// TIA Portal V16 program export: 1 tag tables, 1 data types, 3 data blocks, 9 code blocks (in call order from the OBs), 2 instance data blocks

VAR_GLOBAL   // PLC tag table "Default tag table"
   System_Byte AT %MB1 : Byte;
   FirstScan AT %M1.0 : Bool;
   DiagStatusUpdate AT %M1.1 : Bool;
   AlwaysTRUE AT %M1.2 : Bool;
   AlwaysFALSE AT %M1.3 : Bool;
   Clock_Byte AT %MB0 : Byte;
   Clock_10Hz AT %M0.0 : Bool;
   Clock_5Hz AT %M0.1 : Bool;
   "Clock_2.5Hz" AT %M0.2 : Bool;
   Clock_2Hz AT %M0.3 : Bool;
   "Clock_1.25Hz" AT %M0.4 : Bool;
   Clock_1Hz AT %M0.5 : Bool;
   "Clock_0.625Hz" AT %M0.6 : Bool;
   "Clock_0.5Hz" AT %M0.7 : Bool;
   PositioningAxis_1_Actor_Interface_AddressIn AT %I0.0 : "PD_TEL105_IN";
   PositioningAxis_1_Actor_Interface_AddressOut AT %Q0.0 : "PD_TEL105_OUT";
   PositioningAxis_1_Actor_Interface_TorqueDataAddressIn AT %I40.0 : "PD_TEL750_IN";
   PositioningAxis_1_Actor_Interface_TorqueDataAddressOut AT %Q40.0 : "PD_TEL750_OUT";
   "PositioningAxis_1_Actor_Interface_TorqueDataAddressIn(1)" AT %I44.0 : "PD_TEL750_IN";
   "PositioningAxis_1_Actor_Interface_TorqueDataAddressOut(1)" AT %Q52.0 : "PD_TEL750_OUT";
   SynchronousAxis_1_Actor_Interface_AddressIn AT %I20.0 : "PD_TEL105_IN";
   SynchronousAxis_1_Actor_Interface_AddressOut AT %Q20.0 : "PD_TEL105_OUT";
   SynchronousAxis_1_Actor_Interface_TorqueDataAddressIn AT %I42.0 : "PD_TEL750_IN";
   SynchronousAxis_1_Actor_Interface_TorqueDataAddressOut AT %Q46.0 : "PD_TEL750_OUT";
   "SynchronousAxis_1_Actor_Interface_TorqueDataAddressIn(1)" AT %I46.0 : "PD_TEL750_IN";
   "SynchronousAxis_1_Actor_Interface_TorqueDataAddressOut(1)" AT %Q58.0 : "PD_TEL750_OUT";
END_VAR

TYPE "quad_cnst_array"
// stored: IsFailsafeCompliant false
   STRUCT
      element : Array[0..3, 0..2] of Real;
   END_STRUCT;
   // element[0,0] := 0.00415;   // a
   // element[0,1] := 0.452;   // b
   // element[0,2] := 330.0;   // c
   // element[1,0] := -8.44E-07;   // a
   // element[1,1] := 0.000463;   // b
   // element[1,2] := 0.791;   // c
   // element[2,0] := -9.35E-05;   // a
   // element[2,1] := 0.000775;   // b
   // element[2,2] := 6.34;   // c
   // element[3,0] := -9.04E-05;   // a
   // element[3,1] := 0.0284;   // b
   // element[3,2] := 1.09;   // c
END_TYPE

DATA_BLOCK "testing_purposes"   // DB2
{ S7_Optimized_Access := 'TRUE' }
VERSION : 0.1
// stored: AutoNumber true, DBAccessibleFromOPCUA true, IsOnlyStoredInLoadMemory false, IsRetainMemResEnabled false, IsWriteProtectedInAS false, MemoryReserve 100
   VAR
      emc_calculated : Real;   // EMC_returned
      Temperature : Real := 20.0;   // Chamber temperature [C]
      Air_humi : Real;   // Air humidity [%]
      TemperatureWet : Real := 15.0;   // Wet bulb temperature [C]
      Air_humi_calc : Real;   // Calculated air humidity [%]
      TemperatureWet_calc : Real;   // Calculated wet bulb temperature [C]
      real_sig : Real := 0.0;
      real_win_len : UInt := 20;
      filt_real_sig : Real;
      real_ret_result : Int;   // Real filter work result
      lreal_sig : Real := 0.0;
      lreal_win_len : UInt := 30;
      filt_lreal_sig : Real;
      lreal_ret_result : Int;   // lReal filter work result
   END_VAR
BEGIN
END_DATA_BLOCK

DATA_BLOCK "air_data"   // DB1
{ S7_Optimized_Access := 'TRUE' }
VERSION : 0.1
// stored: AutoNumber true, DBAccessibleFromOPCUA true, IsOnlyStoredInLoadMemory false, IsRetainMemResEnabled false, IsWriteProtectedInAS false, MemoryReserve 100
   VAR RETAIN
      calc_const { S7_SetPoint := 'True'} : "quad_cnst_array";
      Pmean { S7_SetPoint := 'True'} : Real := 1013.25;   // Mean atmospheric pressure [hPa] (mbar)
   END_VAR
BEGIN
END_DATA_BLOCK

DATA_BLOCK "test_blocks_parameters"   // DB4
{ S7_Optimized_Access := 'TRUE' }
VERSION : 0.1
// stored: AutoNumber true, DBAccessibleFromOPCUA true, IsOnlyStoredInLoadMemory false, IsRetainMemResEnabled false, IsWriteProtectedInAS false, MemoryReserve 100
   VAR
      enable : Bool;
      Reset : Bool;
      Restart_to : Bool;
      Home : Bool;
      Settings : Struct
         HomeMode : Int;
      END_STRUCT;
   END_VAR
BEGIN
END_DATA_BLOCK

ORGANIZATION_BLOCK "Main"   // OB1, LAD, ProgramCycle
TITLE = "Main Program Sweep (Cycle)"
{ S7_Optimized_Access := 'TRUE' }
VERSION : 0.1
// stored: AutoNumber true, IsIECCheckEnabled false, SetENOAutomatically false
   VAR_INPUT
      Initial_Call : Bool;   // Initial call of this OB
      Remanence : Bool;   // =True, if remanent data are available
   END_VAR
BEGIN

REGION Network 2 (SCL)
   "test_blocks_DB"();
END_REGION
END_ORGANIZATION_BLOCK

FUNCTION_BLOCK "test_blocks"   // FB2, LAD
{ S7_Optimized_Access := 'TRUE' }
VERSION : 0.1
// stored: AutoNumber true, IsIECCheckEnabled false, IsRetainMemResEnabled false, MemoryReserve 100, SetENOAutomatically false, UDAEnableTagReadback false
   VAR
      MC_POWER_Instance { S7_SetPoint := 'True'} : MC_POWER;
      MC_RESET_Instance { S7_SetPoint := 'True'} : MC_RESET;
      MC_HOME_Instance { S7_SetPoint := 'True'} : MC_HOME;
   END_VAR
BEGIN

REGION Network 1: Enable
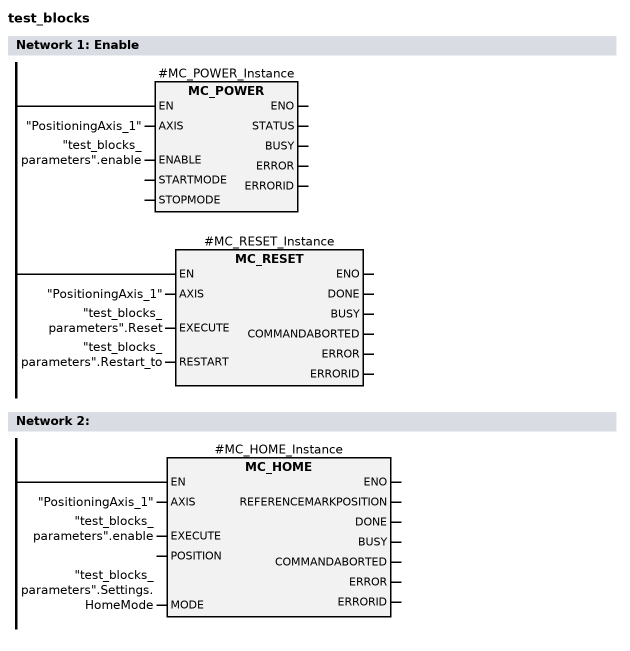
   RUNG wire#powerrail
      #MC_POWER_Instance.MC_POWER(Axis := "PositioningAxis_1", Enable := "test_blocks_parameters".enable, StartMode :=, StopMode :=, Status =>, Busy =>, Error =>, ErrorId =>)
   END_RUNG
   RUNG wire#powerrail
      #MC_RESET_Instance.MC_RESET(Axis := "PositioningAxis_1", Execute := "test_blocks_parameters".Reset, Restart := "test_blocks_parameters".Restart_to, Done =>, Busy =>, CommandAborted =>, Error =>, ErrorId =>)
   END_RUNG
   // the same network as SCL:
   #MC_POWER_Instance(Axis := "PositioningAxis_1", Enable := "test_blocks_parameters".enable);   // MC_POWER
   #MC_RESET_Instance(Axis := "PositioningAxis_1",   // MC_RESET
                      Execute := "test_blocks_parameters".Reset,
                      Restart := "test_blocks_parameters".Restart_to);
END_REGION

REGION Network 2
   RUNG wire#powerrail
      #MC_HOME_Instance.MC_HOME(Axis := "PositioningAxis_1", Execute := "test_blocks_parameters".enable, Position :=, Mode := "test_blocks_parameters".Settings.HomeMode, ReferenceMarkPosition =>, Done =>, Busy =>, CommandAborted =>, Error =>, ErrorId =>)
   END_RUNG
   // the same network as SCL:
   #MC_HOME_Instance(Axis := "PositioningAxis_1",   // MC_HOME
                     Execute := "test_blocks_parameters".enable,
                     Mode := "test_blocks_parameters".Settings.HomeMode);
END_REGION
END_FUNCTION_BLOCK

ORGANIZATION_BLOCK "Cyclic interrupt"   // OB30, LAD, CyclicInterrupt
TITLE = 100ms cyclic interrupt
{ S7_Optimized_Access := 'TRUE' }
VERSION : 0.1
// stored: AutoNumber true, IsIECCheckEnabled false, SetENOAutomatically false
   VAR_INPUT
      Initial_Call : Bool;   // Initial call of this OB
      Event_Count : Int;   // Events discarded
   END_VAR
BEGIN

REGION Network 2
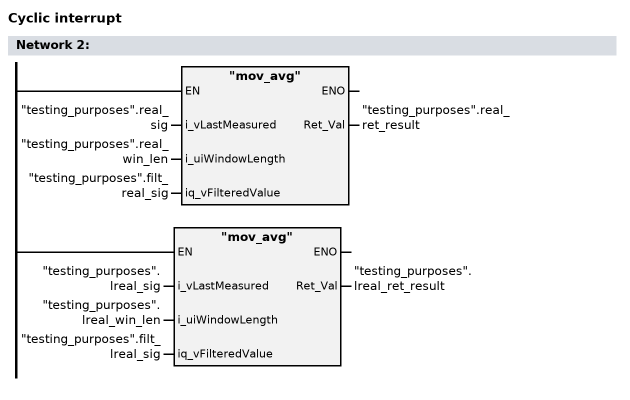
   RUNG wire#powerrail
      "mov_avg"(i_vLastMeasured := "testing_purposes".real_sig, i_uiWindowLength := "testing_purposes".real_win_len, iq_vFilteredValue := "testing_purposes".filt_real_sig, Ret_Val => "testing_purposes".real_ret_result)
   END_RUNG
   RUNG wire#powerrail
      "mov_avg"(i_vLastMeasured := "testing_purposes".lreal_sig, i_uiWindowLength := "testing_purposes".lreal_win_len, iq_vFilteredValue := "testing_purposes".filt_lreal_sig, Ret_Val => "testing_purposes".lreal_ret_result)
   END_RUNG
   // the same network as SCL:
   "testing_purposes".real_ret_result := "mov_avg"(i_vLastMeasured := "testing_purposes".real_sig,
                           i_uiWindowLength := "testing_purposes".real_win_len,
                           iq_vFilteredValue := "testing_purposes".filt_real_sig);
   "testing_purposes".lreal_ret_result := "mov_avg"(i_vLastMeasured := "testing_purposes".lreal_sig,
                           i_uiWindowLength := "testing_purposes".lreal_win_len,
                           iq_vFilteredValue := "testing_purposes".filt_lreal_sig);
END_REGION
END_ORGANIZATION_BLOCK

FUNCTION "mov_avg" : Int
TITLE = Moving average
{ S7_Optimized_Access := 'TRUE' }
AUTHOR : 'A.V.'
VERSION : 0.1
//Simple moving average for signals
   VAR_INPUT 
      i_vLastMeasured : Variant;   // Last measured value for filtering
      i_uiWindowLength : UInt;   // Filter window length
   END_VAR

   VAR_IN_OUT 
      iq_vFilteredValue : Variant;   // Filtered value
   END_VAR

   VAR_TEMP 
      _rStorage : Real;   // Temporary real value for calculations
      _lrStorage : LReal;   // Temporary long real value for calculations
      _rLastMeasured : Real;   // Last measured value of real type
      _lrLastMeasured : LReal;   // Last measured value of long real type
   END_VAR


BEGIN
	#mov_avg := 1;
	// Input and output values must be in same type
	IF TypeOf(#i_vLastMeasured) <> TypeOf(#iq_vFilteredValue)  THEN
	    #mov_avg := -1;
	    RETURN;
	END_IF;
	
	// In case of short window there are no filtering
	IF #i_uiWindowLength < 2 THEN
	    CASE TypeOf(#i_vLastMeasured) OF
	        Real:
	            VariantGet(SRC := #i_vLastMeasured,
	                       DST => #_rStorage);
	            VariantPut(SRC := #_rStorage,
	                       DST := #iq_vFilteredValue);
	        LReal:
	            VariantGet(SRC := #i_vLastMeasured,
	                       DST => #_lrStorage);
	            VariantPut(SRC := #_lrStorage,
	                       DST := #iq_vFilteredValue);
	        ELSE
	            #mov_avg := -1;
	    END_CASE;
	    #mov_avg := 0;
	ELSE
	    CASE TypeOf(#i_vLastMeasured) OF
	        Real:  
	            VariantGet(SRC := #iq_vFilteredValue,
	                       DST => #_rStorage);
	            #_rStorage := #_rStorage * UINT_TO_REAL(#i_uiWindowLength - 1);
	            VariantGet(SRC:=#i_vLastMeasured,
	                       DST=>#_rLastMeasured);
	            #_rStorage := #_rStorage + #_rLastMeasured;
	            #_rStorage := #_rStorage / UINT_TO_REAL(#i_uiWindowLength);
	            VariantPut(SRC:= #_rStorage,
	                       DST:=#iq_vFilteredValue);
	        LReal: 
	            VariantGet(SRC := #iq_vFilteredValue,
	                       DST => #_lrStorage);
	            #_lrStorage := #_lrStorage * UINT_TO_LREAL(#i_uiWindowLength - 1);
	            VariantGet(SRC := #i_vLastMeasured,
	                       DST => #_lrLastMeasured);
	            #_lrStorage := #_lrStorage + #_lrLastMeasured;
	            #_lrStorage := #_lrStorage / UINT_TO_LREAL(#i_uiWindowLength);
	            VariantPut(SRC := #_lrStorage,
	                       DST := #iq_vFilteredValue);;
	        ELSE 
	            #mov_avg := -1;;
	    END_CASE;
	    #mov_avg := 0;
	END_IF;
	
END_FUNCTION

FUNCTION_BLOCK "Main_Safety_RTG1"   // FB1, F_FBD
{ S7_Optimized_Access := 'TRUE' }
VERSION : 0.1
// stored: AutoNumber false, IsIECCheckEnabled false, UDAEnableTagReadback false
BEGIN
END_FUNCTION_BLOCK

FUNCTION "EMC_Calc" : Real
TITLE = Equilibrium moisture content
{ S7_Optimized_Access := 'TRUE' }
AUTHOR : 'A.V. '
VERSION : 0.1
//Function fo calculating Equilibrium moisture content for wood. The Hailwood-Horrobin equation.
   VAR_INPUT 
      T : Real;   // Temperature [C]
      Rh : Real;   // Relative humidity [%]
      cnsts : Array[*, *] of Real;   // Constants for calculation
   END_VAR

   VAR_TEMP 
      Tfh : Real;   // Temperature [Farenheit]
      Rhf : Real;   // Relative humidity [% / 100.0] fractional
      arguments : Array[0..3] of Real;   // Arguments for equation [W, k, k1, k2]
      i : Int;   // row counter
      max_rv_len : DInt;   // Max row index
      max_col_len : DInt;   // Max column index
   END_VAR


BEGIN
	(*
	
	*)
	#Tfh := "LGF_CelsiusToFahrenheit"(#T);
	#Rhf := #Rh / 100.0;
	#max_rv_len := UPPER_BOUND(ARR := #cnsts, DIM := 1);
	#max_col_len := UPPER_BOUND(ARR := #cnsts, DIM := 2);
	FOR #i := 0 TO #max_rv_len DO
	    // Calculating argument values for equation
	    #arguments[#i] := "quad_fnc_value"(x := #Tfh, a := #cnsts[#i, 0], b := #cnsts[#i,1], c := #cnsts[#i,2]);
	END_FOR;
	// Calculating equation value
	#EMC_Calc := (1800.0 / #arguments[0]) * (#arguments[1] * #Rhf / (1 - (#arguments[1] * #Rhf)) + (((#arguments[2]*#arguments[1]*#Rhf) + (2 * #arguments[2] * #arguments[3] * SQR(#arguments[1]) * SQR(#Rhf)))/(1 + (#arguments[2]*#arguments[1]*#Rhf) + (#arguments[2] * #arguments[3] * SQR(#arguments[1]) * SQR(#Rhf)))));
	
END_FUNCTION

FUNCTION "quad_fnc_value" : Real
TITLE = Quadratic function value
{ S7_Optimized_Access := 'TRUE' }
AUTHOR : 'A.V.'
VERSION : 0.1
//Quadraric function value calculation with argument x and constants a, b, c
   VAR_INPUT 
      x : Real;   // Argument
      a : Real;   // Quadratic term constant
      b : Real;   // Linear term constant
      c : Real;   // Free constant
   END_VAR


BEGIN
	(* 
	
	*)
	#quad_fnc_value := (#a * SQR(#x)) + (#b * #x) + #c;
	
END_FUNCTION

FUNCTION "TdRh_Tw" : Real
TITLE = Calculate wet bulb temperature
{ S7_Optimized_Access := 'TRUE' }
AUTHOR : 'A.V.'
VERSION : 0.1
//Function to calculate wet bulb temperature from dry bulb temperature & relative humidity.
   VAR_INPUT 
      Td : Real;   // Dry bulb temperature [C]
      Rh : Real;   // Relative humidity [%]
   END_VAR

   VAR_TEMP 
      Rhf : Real;   // Relative humidity [% / 100.0] fractional
      Tw_iter : Real;   // Running wet bulb temperature for calculations
      Rhc : Real;   // Calculated air relative  humidity [%]
      Ed : Real;   // Saturation vapor pressure in the dry-bulb temperature
      Ew : Real;   // Saturation vapor pressure in the wet-bulb temperature
   END_VAR

   VAR CONSTANT 
      CALC_STEP : Real := 0.1;   // Calculation step size
   END_VAR


BEGIN
	(*
	First approach
	Tw = T * arctan[0.151977 * (RH% + 8.313659)^(1/2)] + arctan(T + RH%) - arctan(RH% - 1.676331) + 0.00391838 *(RH%)^(3/2) * arctan(0.023101 * RH%) - 4.686035.
	Second approach:
	    1) Rhf = (Rh / 100.0%)
	    2) e(d) = 6.112 * EXP[17.62 * Td/(243.12 + Td)]
	    3) e(w) ≈ e(d) * √(Rhf)
	    4) Tw ≈ (237.7 * Log[e(w)/6.108]) / (7.5 - Log[e(w) / 6.108])
	    
	*)
	// First approach calculations
	#TdRh_Tw := #Td * ATAN(0.151977 * (EXP(0.5 * LN(#Rh + 8.313659)))) + ATAN(#Td + #Rh) - ATAN(#Rh - 1.676331) + 0.00391838 * EXP(1.5 * LN(#Rh)) * ATAN(0.023101 * #Rh) - 4.686035;
	// Second approach calculations
	(* // This version doesn't seems to work
	#Rhf := #Rh / 100.0;
	#Ed := 6.112 * EXP(17.502 * #Td / (240.97 + #Td));
	#Ew := #Ed * SQRT(#Rhf);
	#TdRh_Tw := 237.7 * LN(#Ew / 6.108) / (7.5 - LN(#Ew / 6.108));
	*)
	(* 
	#Tw_iter := #Td;
	REPEAT
	    // Iterative calculation of wet bulb temperature
	    #Tw_iter := #Tw_iter - #CALC_STEP;
	    #Rhc := "TdTw_Rh"(Td := #Td, Tw := #Tw_iter, P := "air_data".Pmean);
	UNTIL #Rhc <= #Rh END_REPEAT;
	#TdRh_Tw := #Tw_iter;
	*)
END_FUNCTION

FUNCTION "TdTw_Rh" : Real
TITLE = Calculate relative humidity
{ S7_Optimized_Access := 'TRUE' }
AUTHOR : 'A.V.'
VERSION : 0.1
//Calculate relative humidity from dry bulb temperature & wet bulb temperature
   VAR_INPUT 
      Td : Real;   // Dry bulb temperature [C]
      Tw : Real;   // Wet bulb temperature  [C]
      P : Real;   // Atmospheric pressure [hPa] (mbar)
   END_VAR

   VAR_TEMP 
      A : Real;   // The measuring humidity coefficient
      Ed : Real;   // Saturation vapor pressure in the dry-bulb temperature
      Ew : Real;   // Saturation vapor pressure in the wet-bulb temperature
   END_VAR


BEGIN
	(*
	
	*)
	//Calculating argument values for equation
	#A := 0.00066 * (1 + 0.00115 * #Tw);
	#Ew := 6.112 * EXP(17.502 * #Tw / (240.97 + #Tw));
	#Ed := 6.112 * EXP(17.502 * #Td / (240.97 + #Td));
	#TdTw_Rh := (#Ew - (#A * #P * (#Td - #Tw))) / #Ed * 100.0;
	
END_FUNCTION

DATA_BLOCK "Main_Safety_RTG1_DB"   // DB1, F_DB
NAME : FUSI
VERSION : 0.1
// stored: AutoNumber true, DBAccessibleFromOPCUA true, InstanceOfName Main_Safety_RTG1, InstanceOfType FB
"Main_Safety_RTG1"
BEGIN
END_DATA_BLOCK

DATA_BLOCK "test_blocks_DB"   // DB5
VERSION : 0.1
// stored: AutoNumber true, DBAccessibleFromOPCUA true, InstanceOfName test_blocks, InstanceOfType FB
"test_blocks"
BEGIN
END_DATA_BLOCK
